# EPICS substitutions: EUROTHRM/EUROTHRM-IOC-01App/Db/devEurothrmA06.substitutions
# Note: this file is generated by generate_substitutions.py
file devEurothrm.template {
pattern { P, GAD, LAD, MODBUS_PV, MODBUS_SP, MODBUS_P, MODBUS_I, MODBUS_D, MODBUS_HS, MODBUS_LS, MODBUS_AT, MODBUS_HO, MODBUS_OP }
{ "\$(P)", "0", "6", "5121", "5122", "5126", "5128", "5129", "5231", "5232", "5390", "5150", "5123" }
}
